(* IEC 61131-3 sources: IceManRemastered/Device/application/Control, 3 files *)

(* ---- MotionCommand.st ---- *)
TYPE MotionCommand :
STRUCT
	Steps: UDINT;
	Direction: UINT;
	Speed: UINT;
END_STRUCT
END_TYPE

(* ---- Control.gvl.st ---- *)
{attribute 'qualified_only'}
VAR_GLOBAL
	FaultReset: FaultReset;
	Logger: Logger;
	ManualControl: ManualControl;
	LoadDefaults: BOOL;
END_VAR

(* ---- TempConditioner.st ---- *)
FUNCTION TempConditioner : REAL
VAR_INPUT
	TempInput: 			UINT;				//
END_VAR
VAR
END_VAR

// --- BEGIN IMPLEMENTATION ---

TempConditioner := UINT_TO_REAL(TempInput) / 10;
